TYPE ST_MoverParams :
STRUCT
	lrVelocity		: LREAL ;
	lrVelocity_c	: LREAL ;
END_STRUCT
END_TYPE

(* stored: Version 1.1.0.1
   DUT ST_MoverParams: Id {140ebeae-1a01-465a-b83d-adf54988880b} *)
